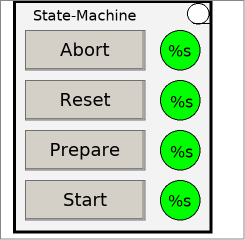
VISUALIZATION StarterKitStateMachinelPad  // 245x240
VAR_IN_OUT
	
	stControlPadControl		:   ST_Vis_ControlPadControl;

END_VAR
    Rectangle (13,0 199x233)
    Button (25,30 120x40), "Abort"
        tap stControlPadControl.bButtonState_Abort p3779583253=TRUE
    Button (25,80 120x40), "Reset"
        tap stControlPadControl.bButtonState_Reset
    Button (25,130 120x40), "Prepare"
        tap stControlPadControl.bButtonState_Prepare
    Button (25,180 120x40), "Start"
        tap stControlPadControl.bButtonState_Start
    Ellipse (160,30 40x40)
    Ellipse (160,30 40x40), invisible if: NOT stControlPadControl.bStateSignalAbortYellow
    Group (160,80 40x40)
        Ellipse (0,0 40x40)
        Ellipse (0,0 40x40), invisible if: NOT stControlPadControl.bStateSignalResetYellow
        Ellipse (0,0 40x40), invisible if: NOT stControlPadControl.bStateSignalResetGreen
    Group (160,130 40x40)
        Ellipse (0,0 40x40)
        Ellipse (0,0 40x40), invisible if: NOT stControlPadControl.bStateSignalPrepareYellow
        Ellipse (0,0 40x40), invisible if: NOT stControlPadControl.bStateSignalPrepareGreen
    Group (160,180 40x40)
        Ellipse (0,0 40x40)
        Ellipse (0,0 40x40), invisible if: NOT stControlPadControl.bStateSignalExecuteYellow
        Ellipse (0,0 40x40), invisible if: NOT stControlPadControl.bStateSignalExecuteGreen
    Ellipse (160,30 40x40), invisible if: NOT stControlPadControl.bStateSignalAbortBlue
    Ellipse (160,30 40x40), invisible if: NOT stControlPadControl.bStateSignalAbortGreen
    Label (19,1 132x29), "State-Machine"
    Textfield (159,35 42x32), "%s", text variable: stControlPadControl.iAbortSequenceState, invisible if: stControlPadControl.bAbortSequenceStateInvisible
    Textfield (161,86 42x32), "%s", text variable: stControlPadControl.iResetSequenceState, invisible if: stControlPadControl.bResetSequenceStateInvisible
    Textfield (161,136 42x32), "%s", text variable: stControlPadControl.iPrepareSequenceState, invisible if: stControlPadControl.bPrepareSequenceStateInvisible
    Textfield (159,185 42x32), "%s", text variable: stControlPadControl.iStartSequenceState, invisible if: stControlPadControl.bStartSequenceStateInvisible
    Ellipse (187,3 22x21)
    Line (230,-7) (245,-6)
    Line (193,23) (209,23)
    Rectangle (179,3 32x25)
        OnMouseClick: execute { stControlPadControl.bVisInvisibleButton := TRUE; }
END_VISUALIZATION

(* stored: Version 1.1.0.1
   Visu StarterKitStateMachinelPad: Id {56dcc308-0024-42b9-b3a9-6120f95e25f2} *)
